Yaskawa INFORM job: FRONT_SEARCH_-90ST-1_5240.JBI

/JOB
//NAME FRONT_SEARCH_-90ST-1_5240
///FOLDERNAME 02-SKRZYNIE_JOBS
//POS
///NPOS 28,28,0,6,0,0
///TOOL 0
///POSTYPE PULSE
///PULSE
C00000=-1,-11355,44471,-89821,-32839,-4429
C00001=42981,-20293,9138,-37936,728,-21145
C00002=54060,-18370,-3633,-35664,24175,-28224
C00003=52297,-12132,7037,-37532,21360,-27406
C00004=51942,-10733,9481,-38131,20724,-27135
C00005=51077,-9689,10456,-36945,20459,-27806
C00006=51301,-9073,12804,-39146,19655,-26685
C00007=51942,-10733,9481,-38131,20724,-27135
C00008=18711,-22105,1064,-162831,-11969,28252
C00009=18711,-22105,1064,-162831,-11969,28252
C00010=18532,-21440,1557,-162623,-12145,28140
C00011=18637,-20703,4198,-161579,-10900,27647
C00012=18711,-22105,1064,-162831,-11969,28252
C00013=-17436,-23335,-3703,-127893,-26127,3675
C00014=-17436,-23335,-3703,-127893,-26127,3675
C00015=-17154,-22427,-3036,-128420,-26139,3977
C00016=-17249,-21945,-1001,-126803,-25497,3120
C00017=-17436,-23335,-3703,-127893,-26127,3675
C00018=-19623,-34877,-16768,-124729,-29078,-51940
C00019=-20248,-24303,-1312,-151363,-11605,-35820
C00020=-19804,-24319,-727,-151735,-11109,-35599
C00021=-19430,-23337,-33,-153249,-11256,-34838
C00022=-19543,-22852,1896,-151010,-10397,-35920
C00023=-19804,-24319,-727,-151735,-11109,-35599
C00024=-22935,-43287,-23487,-146875,-13252,-38235
C00025=-53252,-41973,-2905,-102185,-37459,-42403
C00026=0,-35574,42087,-36666,-9339,-1809
C00027=0,-52278,40443,0,6873,1
BC00000=889812
BC00001=985413
BC00002=985413
BC00003=985413
BC00004=985413
BC00005=985413
BC00006=985413
BC00007=985413
BC00008=985414
BC00009=985414
BC00010=985414
BC00011=985414
BC00012=985414
BC00013=985413
BC00014=985413
BC00015=985413
BC00016=985413
BC00017=985413
BC00018=985413
BC00019=985413
BC00020=985413
BC00021=985413
BC00022=985413
BC00023=985413
BC00024=972047
BC00025=926709
BC00026=812358
BC00027=805481
///POSTYPE BASE
///RECTAN
///RCONF 0,0,0,0,0,0,0,0,0,0,0,0,0,0,0,0,0,0,0,0,0,0,0,0
P00006=-2.449,0.031,8.825,0.0000,0.0000,0.0000
P00058=0.000,0.000,3.000,0.0000,0.0000,0.0000
P00501=-2.026,0.009,3.534,0.0000,0.0000,0.0000
///RCONF 1,0,0,0,0,0,0,0,0,0,0,0,0,0,0,0,0,0,0,0,0,0,0,0
P00502=-2.023,0.001,1.732,0.0000,0.0000,0.0000
P00503=0.138,-0.044,1.539,0.0000,0.0000,0.0000
P00504=-0.309,-0.010,1.636,0.0000,0.0000,0.0000
//INST
///DATE 2024/05/18 20:52
///ATTR SC,RW
///GROUP1 RB1,BS1
NOP
MOVJ C00000 BC00000 VJ=40.00
'::::::::::::::::::::::::::::::::
'W56 P
'::::::::::::::::::::::::::::::::
MOVL C00001 BC00001 V=500.0
MOVL C00002 BC00002 V=500.0
MOVL C00003 BC00003 V=500.0
MOVL C00004 BC00004 V=166.7 PL=0
REFP 3 C00005 BC00005
CALL JOB:SEARCH-R1
IMOV P0058 V=23.0
SET P0501 P0006
SFTON P0501
REFP 3 C00006 BC00006
CALL JOB:SEARCH-R1
SET P0501 P0006
SFTON P0501
MOVL C00007 BC00007 V=166.7 PL=0
SFTOF
'::::::::::::::::::::::::::::::::
'W56 L
'::::::::::::::::::::::::::::::::
MOVL C00008 BC00008 V=333.3
MOVL C00009 BC00009 V=166.7 PL=0
REFP 3 C00010 BC00010
CALL JOB:SEARCH-R1
IMOV P0058 V=23.0
SET P0502 P0006
SFTON P0502
REFP 3 C00011 BC00011
CALL JOB:SEARCH-R1
SET P0502 P0006
SFTON P0502
MOVL C00012 BC00012 V=166.7 PL=0
SFTOF
'::::::::::::::::::::::::::::::::
'W57 P
'::::::::::::::::::::::::::::::::
MOVL C00013 BC00013 V=250.0
MOVL C00014 BC00014 V=166.7 PL=0
REFP 3 C00015 BC00015
CALL JOB:SEARCH-R1
IMOV P0058 V=23.0
SET P0503 P0006
SFTON P0503
REFP 3 C00016 BC00016
CALL JOB:SEARCH-R1
SET P0503 P0006
SFTON P0503
MOVL C00017 BC00017 V=250.0 PL=0
SFTOF
'::::::::::::::::::::::::::::::::
'W57 L
'::::::::::::::::::::::::::::::::
MOVL C00018 BC00018 V=333.3
MOVL C00019 BC00019 V=333.3
MOVL C00020 BC00020 V=166.7 PL=0
REFP 3 C00021 BC00021
CALL JOB:SEARCH-R1
IMOV P0058 V=23.0
SET P0504 P0006
SFTON P0504
REFP 3 C00022 BC00022
CALL JOB:SEARCH-R1
SET P0504 P0006
SFTON P0504
MOVL C00023 BC00023 V=166.7 PL=0
SFTOF
MOVJ C00024 BC00024 VJ=40.00
MOVJ C00025 BC00025 VJ=50.00
MOVJ C00026 BC00026 VJ=50.00
MOVJ C00027 BC00027 VJ=50.00
END
